{attribute addProperty BoxType "KL9900-0064"}
{attribute addProperty Id "Channel_1Channel_7B6F5FAF00"}
{attribute addProperty CRC "2977761574"}
{attribute addProperty SizeInBites "0"}
{attribute addProperty SizeInBytes "0"}
TYPE KL_B17D0926 :
STRUCT
	{attribute addProperty Name "Channel_1"}
	Channel_1 : Channel_7B6F5FAF;
END_STRUCT
END_TYPE

(* stored: Version 1.2.0.0, ProductVersion 3.1.4024.9
   DUT KL_B17D0926: Id {fddd43ec-ca21-4de5-9f47-0167c0f31f0b} *)
